RoboDK station: 2E06666.rdk

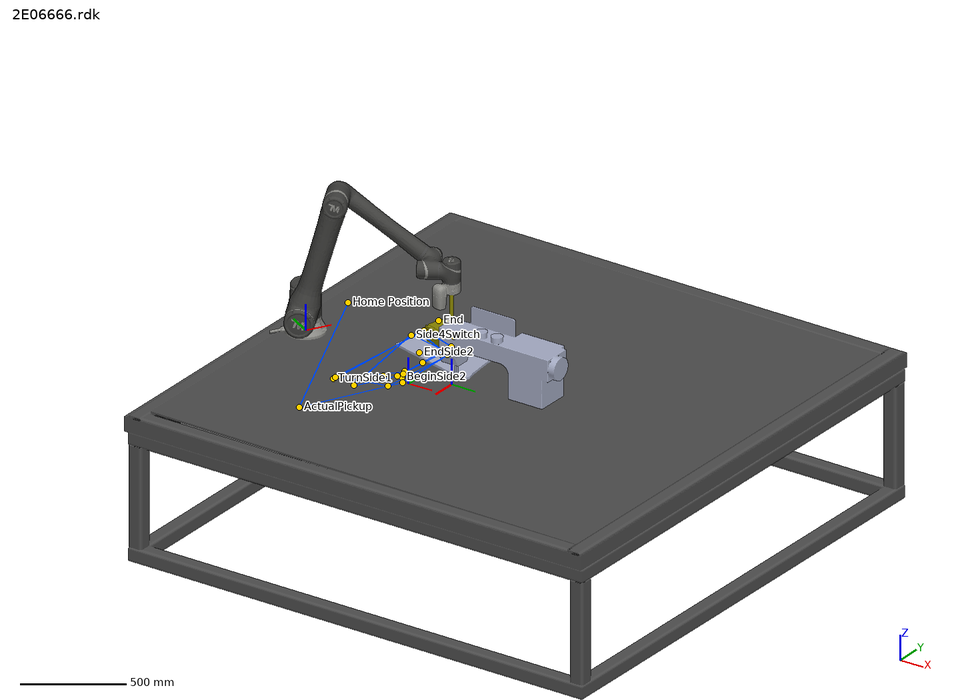
[picture v0: the station drawn from its stored meshes, robots at their saved joint values, targets as dots, program paths as lines]
Station 2E06666VentacPiece_Side1n2n3n4_220421 (saved by RoboDK 5.2.0). Poses are relative to the parent item; angles as X-Y-Z fixed-axis rotations.
Station parameters (name, value as stored): IO_5, 40, OPC-UA, opc.tcp://localhost:4840
  - frame Omron TM12 Base at (190, -120, 780) mm, rotated rx 0 ry 0 rz 60 deg
    - robot Omron TM12: 6 axes, payload 12 kg, reach 1300 mm, repeatability 0.1 mm, weight 33.3 kg
        modified DH rows (alpha deg, a mm, theta deg, d mm): 0, 0, 0, 165.2; 90, 0, 90, 0; 0, 636.1, 0, 0; 0, 557.9, -90, 156.3; -90, 0, 0, 106; 90, 0, 180, 113.15
        base shift (0.29, 0, -5.5) mm
        joint limits [-270, -180, -166, -180, -180, -270] to [270, 180, 166, 180, 180, 270]; home [0, 0, 90, 0, 90, 0]; saved at [-31.982, 15.329, 112.788, -37.754, 90.568, 133.439]
      - tool KVG-gripper, TCP at (0, 0, 285) mm, size 287.4 x 120 x 282 mm, geometry from untitled.obj
        - object 2E06666_REV_C - Copy2 at (18.39, 14.06, 15.2) mm, rotated rx -180 ry 0 rz -91.02 deg, size 361.2 x 491.2 x 12 mm, geometry from 2E06666_REV_C - Copy2.IGS
    - target Home Position (Cartesian target) at (-0.43, -475.84, 354) mm, rotated rx -178.71 ry -1.76 rz 148.98 deg; joints [-69.005, -0.122, 95.32, 175.401, -87.9, 52.005] of Omron TM12
    - target ActualPickup (Cartesian target) at (-394.64, -777.36, 21.11) mm, rotated rx -177.4 ry 0.83 rz -152.95 deg; joints [-107.727, 26.497, 97.569, -35.328, 92.42, -224.731] of Omron TM12
    - target TurnSide1 (Cartesian target) at (-131.33, -594.7, 35) mm, rotated rx -179.74 ry 0.68 rz -61.29 deg; joints [-87.533, 22.491, 102.653, 145.583, -89.927, -116.244] of Omron TM12
    - target BeginSide2 (Cartesian target) at (168.67, -714.7, 35) mm, rotated rx -179.74 ry 0.68 rz -66.29 deg; joints [91.005, -16.051, -111.762, 37.083, -90.028, 67.294] of Omron TM12
    - target EndSide2 (Cartesian target) at (358.67, -504.7, 30) mm, rotated rx -179.74 ry 0.68 rz -61.29 deg; joints [110.648, -6.61, -123.864, 39.761, -89.842, 81.935] of Omron TM12
    - target End (Cartesian target) at (579.33, -246.94, 38.32) mm, rotated rx -178.91 ry 0.4 rz 61.35 deg; joints [-8.72, 7.16, 122, -38, 90, 19.93] of Omron TM12
    - target Target 7 (Cartesian target) at (168.67, -714.7, 35) mm, rotated rx -179.74 ry 0.68 rz -66.29 deg; joints [-64.606, 15.727, 111.514, -36.564, 90.276, 91.681] of Omron TM12
    - target CurrentPosition (Cartesian target) at (95.48, -662.89, 34.03) mm, rotated rx -179.84 ry 0.65 rz -95.42 deg; joints [-68.6, 10.56, 118.55, -38.6, 90.44, 116.82] of Omron TM12
    - target BeginSide2. (Cartesian target) at (206.92, -665.73, 35) mm, rotated rx -179.87 ry 0.95 rz -77.8 deg; joints [-60.04, 12.869, 115.345, -37.344, 90.411, -252.239] of Omron TM12
    - target Midside2 (Cartesian target) at (325.48, -612.89, 34.03) mm, rotated rx -179.84 ry 0.65 rz -80.42 deg; joints [-49.312, 28.838, 91.958, 149.679, -90.477, -58.892] of Omron TM12
    - target EndSide2 (Cartesian target) at (522.31, -505.58, 30) mm, rotated rx -179.84 ry 0.65 rz -75.42 deg; joints [-31.982, 15.329, 112.788, -37.754, 90.568, 133.439] of Omron TM12
    - target MoveTo3 (Cartesian target) at (-89.18, -583.7, 34.03) mm, rotated rx -179.84 ry 0.65 rz 29.58 deg; joints [-82.9, 3.387, 127.166, -40.652, 89.333, -22.479] of Omron TM12
    - target Start3 (Cartesian target) at (70.15, -772.41, 34.03) mm, rotated rx -179.84 ry 0.65 rz 29.58 deg; joints [-72.852, 18.627, 107.674, -36.283, 89.326, -12.43] of Omron TM12
    - target EndSide3 (Cartesian target) at (486.02, -572.72, 30) mm, rotated rx -179.84 ry 0.65 rz 29.58 deg; joints [-37.393, 17.119, 110.266, -36.98, 89.462, 23.03] of Omron TM12
    - target Side4Switch (Cartesian target) at (399.57, -324.95, 34.03) mm, rotated rx -179.84 ry 0.65 rz 124.58 deg; joints [-21.055, -3.912, 134.502, -41.038, 89.496, -55.635] of Omron TM12
    - target Side4 (Cartesian target) at (-74.15, -698.58, 34.03) mm, rotated rx -179.84 ry 0.65 rz 119.58 deg; joints [-83.288, 12.671, 116.104, -39.44, 90.104, -112.866] of Omron TM12
    - target BeginSide4 (Cartesian target) at (155.73, -692.6, 34.03) mm, rotated rx -179.84 ry 0.65 rz 116.05 deg; joints [-64.54, 13.227, 115.363, -39.245, 89.844, -90.59] of Omron TM12
    - target EndSide4 (Cartesian target) at (477.5, -549.92, 34.03) mm, rotated rx -179.84 ry 0.65 rz 116.05 deg; joints [-36.403, 14.709, 113.324, -38.538, 89.553, -62.454] of Omron TM12
    - target Release (Cartesian target) at (576.89, -422.07, 34.03) mm, rotated rx -179.84 ry 0.65 rz 119.58 deg; joints [-23.27, 29.808, 90.162, 149.606, -89.475, 127.15] of Omron TM12
    - target BeginSide1 (Cartesian target) at (157.15, -752.2, 25) mm, rotated rx -179.87 ry 0 rz -150 deg; joints [-66.491, 18.599, 108.905, -37.629, 90.014, -186.491] of Omron TM12
    - target EndSide1 (Cartesian target) at (473.75, -569.41, 25.16) mm, rotated rx -179.79 ry 0.94 rz -150 deg; joints [-38.51, 16.353, 112.212, -39.099, 90.797, -158.504] of Omron TM12
    - target Mid (Cartesian target) at (447.33, -323.61, 35) mm, rotated rx -179.87 ry 0.95 rz -122.8 deg; joints [-20.127, -0.053, 130.687, -40.967, 90.903, 192.68] of Omron TM12
    - target Mid2 (Cartesian target) at (-119.01, -587.8, 35) mm, rotated rx -179.87 ry 0.95 rz -62.8 deg; joints [-86.187, 4.676, 125.359, -39.11, 89.737, 66.62] of Omron TM12
    - target Target 24 (Cartesian target) at (192.09, -683.61, 34.03) mm, rotated rx -179.84 ry 0.65 rz -80.42 deg; joints [-61.819, 13.826, 114.264, -37.522, 90.363, -251.399] of Omron TM12
    - target Mid3 (Cartesian target) at (479.99, -296.92, 30) mm, rotated rx -179.84 ry 0.65 rz -80.42 deg; joints [-16.156, 18.683, 108.145, 143.309, -90.66, -25.735] of Omron TM12
  - frame Tool at (0, 1000, 0) mm
    - object Machine at (1443.88, -1066.05, 820) mm, rotated rx 0 ry 0 rz -90 deg, size 180 x 665 x 356.6 mm, geometry from Machine.IGS
  - object Table 108x114x32 IN at (0, 0, 0) mm, size 2628.9 x 2679.7 x 778.4 mm, geometry from Table-108x114x32-IN.sld
  - program Prog1 (27 instructions, listed below)
  - frame Needle at (1090, -200, 780) mm, rotated rx 0 ry 0 rz -90 deg
  - object 208553A at (130, 0, 400) mm, rotated rx 10 ry 0 rz 0 deg, size 459 x 478.2 x 12 mm, geometry from 208553A.IGS
  - object 30128608- at (0, 0, 0) mm, size 802 x 205 x 30 mm, geometry from 30128608-.IGS
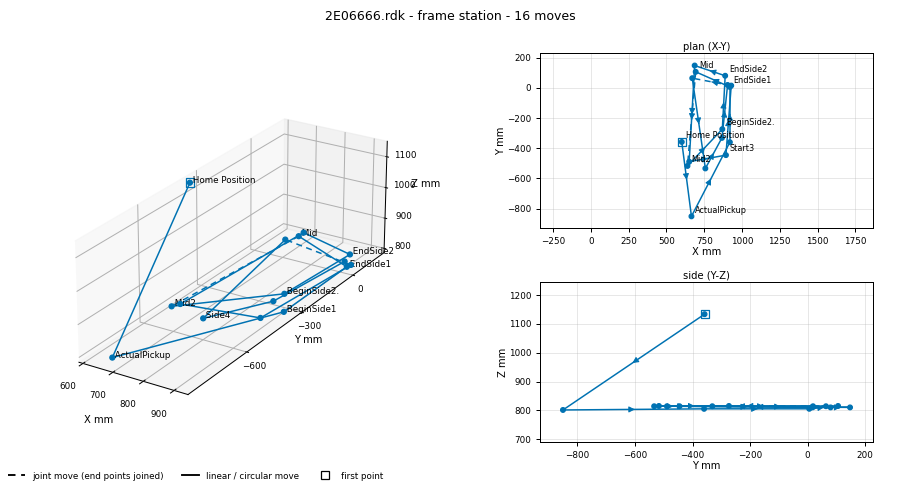
[picture p0: tool path of 2E06666.rdk in frame station, 16 of 16 moves have a stored position in this frame; points joined in program order, loops and branches not executed]

--- program Prog1 (robot Omron TM12) ---
  Set Ref.: Omron TM12 Base
  Set Tool: KVG-gripper
  MoveL (Home Position)
  MoveL (ActualPickup)
  Set IO_5=40
  MoveL (BeginSide1)
  Set IO_5=20
  MoveL (EndSide1)
  Set IO_5=30
  MoveL (Mid)
  MoveJ (Mid2)
  MoveL (BeginSide2.)
  Set IO_5=20
  MoveL (EndSide2)
  Set IO_5=30
  MoveL (Mid3)
  MoveL (MoveTo3)
  MoveL (Start3)
  Set IO_5=20
  MoveL (EndSide3)
  Set IO_5=30
  MoveJ (Side4Switch)
  MoveL (Side4)
  MoveL (BeginSide4)
  Set IO_5=20
  MoveL (EndSide4)
  Set IO_5=30
